// TwinCAT 3 PLC project test
// ProgramVersion: 3.1.4020.5
// libraries:
//   L2Si Vacuum Library, * (SLAC)
//   Tc2_Standard, * (Beckhoff Automation GmbH)
//   Tc2_System, * (Beckhoff Automation GmbH)
//   Tc3_Module, * (Beckhoff Automation GmbH)
// project tree:
//   GVLs/ GVL_Devices.TcGVL (not stored)
//   / PlcTask.TcTTO (not stored)
//   POUs/ MAIN.TcPOU
// real-time tasks:
//   TASK PlcTask: cycle T#10ms, priority 20, ADS port 350
// I/O:
//   DEVICE Device 1 (EtherCAT) (disabled), AmsNetId 5.40.55.128.2.1
//     Term 1 (EK1100) [EK1100 EtherCAT Coupler (2A E-Bus)]
//       Term 2 (EL3174-0002) [EL3174-0002 4Ch. Ana. Input +/-10V, +/-20mA 16 Bit, Isolated Channels]
//       Term 3 (EL3174-0002) [EL3174-0002 4Ch. Ana. Input +/-10V, +/-20mA 16 Bit, Isolated Channels]
//       Term 4 (EL2624) [EL2624 4Ch. Relay Output, NO (125V AC / 30V DC)]
//       Term 6 (EL1004) [EL1004 4Ch. Dig. Input 24V, 3ms]
//       Term 5 (EL1004) [EL1004 4Ch. Dig. Input 24V, 3ms]
//       Term 7 (EL2004) [EL2004 4Ch. Dig. Output 24V, 0.5A]
//       Term 8 (EL3064) [EL3064 4Ch. Ana. Input 0-10V]
//       Term 9 (EL2794) [EL2794 4Ch. Dig. Output 24V AC/DC, 2A, short-circuit-proof]
//       Term 10 (EL1004) [EL1004 4Ch. Dig. Input 24V, 3ms]
//       Term 11 (EL1124) [EL1124 4Ch. Dig. Input 5V, 10µs, Sensor Power]
//       Term 12 (EL1124) [EL1124 4Ch. Dig. Input 5V, 10µs, Sensor Power]
//       Term 13 (EL3064) [EL3064 4Ch. Ana. Input 0-10V]
// variable links:
//   SIM/SIM Instance <-> test/test Instance
//     PlcTask Inputs/GVL_SimDevices.S_FEE_GCC_03.i_xHvOn <-> PlcTask Outputs/GVL_Devices.FEE_GCC_03.q_xHV_DIS
//     PlcTask Inputs/GVL_SimDevices.S_FEE_GCC_04.i_xHvOn <-> PlcTask Outputs/GVL_Devices.FEE_GCC_04.q_xHV_DIS
//     PlcTask Inputs/GVL_SimDevices.S_FEE_KMONO_GCC_01.i_xHvOn <-> PlcTask Outputs/GVL_Devices.FEE_KMONO_GCC_01.q_xHV_DIS
//     PlcTask Inputs/GVL_SimDevices.S_FEE_KMONO_PIP_01.xOn <-> PlcTask Outputs/GVL_Devices.FEE_KMONO_PIP_01.q_xHVEna_DO
//     PlcTask Inputs/GVL_SimDevices.S_FEE_M1L_PIP_01.xOn <-> PlcTask Outputs/GVL_Devices.FEE_M1L_PIP_01.q_xHVEna_DO
//     PlcTask Inputs/GVL_SimDevices.S_FEE_MIL_GCC_02.i_xHvOn <-> PlcTask Outputs/GVL_Devices.FEE_M1L_GCC_01.q_xHV_DIS
//     PlcTask Inputs/GVL_SimDevices.S_FEE_PIP_02.xOn <-> PlcTask Outputs/GVL_Devices.FEE_PIP_02.q_xHVEna_DO
//     PlcTask Inputs/GVL_SimDevices.S_FEE_PIP_03.xOn <-> PlcTask Outputs/GVL_Devices.FEE_PIP_03.q_xHVEna_DO
//     PlcTask Inputs/GVL_SimDevices.S_FEE_VGC_02.i_xSol <-> PlcTask Outputs/GVL_Devices.FEE_VGC_02.q_xOPN_DO
//     PlcTask Inputs/GVL_SimDevices.S_FEE_VGC_03.i_xSol <-> PlcTask Outputs/GVL_Devices.FEE_VGC_03.q_xOPN_DO
//     PlcTask Inputs/GVL_SimDevices.S_FEE_VGC_04.i_xSol <-> PlcTask Outputs/GVL_Devices.FEE_VGC_04.q_xOPN_DO
//     PlcTask Outputs/GVL_SimDevices.S_FEE_GCC_03.q_DisActive <-> PlcTask Inputs/GVL_Devices.FEE_GCC_03.i_xDisc_Active
//     PlcTask Outputs/GVL_SimDevices.S_FEE_GCC_04.q_DisActive <-> PlcTask Inputs/GVL_Devices.FEE_GCC_04.i_xDisc_Active
//     PlcTask Outputs/GVL_SimDevices.S_FEE_GCC_03.q_iRawPress <-> PlcTask Inputs/GVL_Devices.FEE_GCC_03.i_iPRESS_R
//     PlcTask Outputs/GVL_SimDevices.S_FEE_GCC_04.q_iRawPress <-> PlcTask Inputs/GVL_Devices.FEE_GCC_04.i_iPRESS_R
//     PlcTask Outputs/GVL_SimDevices.S_FEE_GCC_03.q_xHVOn <-> PlcTask Inputs/GVL_Devices.FEE_GCC_03.i_xHV_ON
//     PlcTask Outputs/GVL_SimDevices.S_FEE_GCC_04.q_xHVOn <-> PlcTask Inputs/GVL_Devices.FEE_GCC_04.i_xHV_ON
//     PlcTask Outputs/GVL_SimDevices.S_FEE_GPI_03.q_iRawPress <-> PlcTask Inputs/GVL_Devices.FEE_GPI_03.i_iPRESS_R
//     PlcTask Outputs/GVL_SimDevices.S_FEE_GPI_04.q_iRawPress <-> PlcTask Inputs/GVL_Devices.FEE_GPI_04.i_iPRESS_R
//     PlcTask Outputs/GVL_SimDevices.S_FEE_KMONO_GCC_01.q_DisActive <-> PlcTask Inputs/GVL_Devices.FEE_KMONO_GCC_01.i_xDisc_Active
//     PlcTask Outputs/GVL_SimDevices.S_FEE_KMONO_GCC_01.q_iRawPress <-> PlcTask Inputs/GVL_Devices.FEE_KMONO_GCC_01.i_iPRESS_R
//     PlcTask Outputs/GVL_SimDevices.S_FEE_KMONO_GCC_01.q_xHVOn <-> PlcTask Inputs/GVL_Devices.FEE_KMONO_GCC_01.i_xHV_ON
//     PlcTask Outputs/GVL_SimDevices.S_FEE_KMONO_GPI_01.q_iRawPress <-> PlcTask Inputs/GVL_Devices.FEE_KMONO_GPI_01.i_iPRESS_R
//     PlcTask Outputs/GVL_SimDevices.S_FEE_M1L_GPI_02.q_iRawPress <-> PlcTask Inputs/GVL_Devices.FEE_M1L_GPI_01.i_iPRESS_R
//     PlcTask Outputs/GVL_SimDevices.S_FEE_MIL_GCC_02.q_DisActive <-> PlcTask Inputs/GVL_Devices.FEE_M1L_GCC_01.i_xDisc_Active
//     PlcTask Outputs/GVL_SimDevices.S_FEE_MIL_GCC_02.q_iRawPress <-> PlcTask Inputs/GVL_Devices.FEE_M1L_GCC_01.i_iPRESS_R
//     PlcTask Outputs/GVL_SimDevices.S_FEE_MIL_GCC_02.q_xHVOn <-> PlcTask Inputs/GVL_Devices.FEE_M1L_GCC_01.i_xHV_ON
//     PlcTask Outputs/GVL_SimDevices.S_FEE_VGC_02.q_xClsLS <-> PlcTask Inputs/GVL_Devices.FEE_VGC_02.i_xClsLS
//     PlcTask Outputs/GVL_SimDevices.S_FEE_VGC_03.q_xClsLS <-> PlcTask Inputs/GVL_Devices.FEE_VGC_03.i_xClsLS
//     PlcTask Outputs/GVL_SimDevices.S_FEE_VGC_04.q_xClsLS <-> PlcTask Inputs/GVL_Devices.FEE_VGC_04.i_xClsLS
//     PlcTask Outputs/GVL_SimDevices.S_FEE_VGC_02.q_xOpnLS <-> PlcTask Inputs/GVL_Devices.FEE_VGC_02.i_xOpnLS
//     PlcTask Outputs/GVL_SimDevices.S_FEE_VGC_03.q_xOpnLS <-> PlcTask Inputs/GVL_Devices.FEE_VGC_03.i_xOpnLS
//     PlcTask Outputs/GVL_SimDevices.S_FEE_VGC_04.q_xOpnLS <-> PlcTask Inputs/GVL_Devices.FEE_VGC_04.i_xOpnLS

// ---- POUs/MAIN.TcPOU
PROGRAM MAIN
VAR

END_VAR


//valves
FEE_VGC_02(i_stUSG := , i_stDSG:= FEE_KMONO_GCC_01.IG, i_xDis_DPIlk:= FALSE, i_xEPS_OK:= TRUE, i_xPMPS_OK:= TRUE);
FEE_VGC_03(i_stUSG := FEE_KMONO_GCC_01.IG, i_stDSG:= FEE_M1L_GCC_01.IG, i_xDis_DPIlk:= FALSE, i_xEPS_OK:= TRUE, i_xPMPS_OK:= TRUE);
FEE_VGC_04(i_stUSG :=FEE_GCC_03.IG , i_stDSG:= , i_xDis_DPIlk:= FALSE, i_xEPS_OK:= TRUE, i_xPMPS_OK:= TRUE);

// gauges and pip
FEE_KMONO_GPI_01(PG=>);
FEE_KMONO_GCC_01(PG:=FEE_KMONO_GPI_01.PG);
FEE_KMONO_PIP_01(i_stGauge:= FEE_KMONO_GCC_01.IG);

FEE_GPI_03(PG=>);
FEE_GCC_03(PG:=FEE_KMONO_GPI_01.PG);

FEE_PIP_02(i_stGauge:= FEE_GCC_03.IG);

FEE_M1L_GPI_01(PG=>);
FEE_M1L_GCC_01(PG:=FEE_M1L_GPI_01.PG);
FEE_M1L_PIP_01(i_stGauge:= FEE_M1L_GCC_01.IG);

FEE_GPI_04(PG=>);
FEE_GCC_04(PG:=FEE_GPI_04.PG);
FEE_PIP_03(i_stGauge:= FEE_GCC_04.IG);

END_PROGRAM
